FUNCTION_BLOCK FB_Joystick_Input_Scaling
VAR_INPUT
<<<<<<< HEAD
	nRawInput : INT; 
	stJoystickInputScaling : ST_JoystickInputScaling;
	eStatus : E_Status := E_Status.Checking; // bEnable erstatter
=======
	bEnable : BOOL;
	nRawInput : INT; 
	stJoystickInputScaling : ST_JoystickInputScaling;
>>>>>>> 39be3fc96e305d29936f65dffbbc69267e7bf2cf
END_VAR
VAR_OUTPUT
	fNormalizedOutput : LREAL; 
END_VAR
VAR
	fRawInput : LREAL;
	fTempInput : LREAL;
	fTempOutput : LREAL; 
END_VAR

fRawInput := INT_TO_LREAL(nRawInput); // konverterer heltallsverdi fra joystick til flyt-verdi, for beregninger med desimaltall

fTempInput := fRawInput - stJoystickInputScaling.fNeutralInputValue; //Midlertidig variabel før normalisering, midtstilling får en verdi nær 0

IF fTempInput > stJoystickInputScaling.fNeutralDeadband THEN
	fTempOutput := fTempInput/(stJoystickInputScaling.fMaxInputValue - stJoystickInputScaling.fNeutralInputValue);	// Normalisert verdi mellom 0 og 1

ELSIF	fTempInput < -stJoystickInputScaling.fNeutralInputValue THEN 
	fTempOutput := fTempInput/(stJoystickInputScaling.fMaxInputValue - stJoystickInputScaling.fNeutralInputValue); // Normalisert vedi mellom 0 og -1
	
ELSE	
    fTempOutput := 0.0;
END_IF

<<<<<<< HEAD
IF eStatus = E_status.Running AND G_IO.bManualSwitch THEN
=======
IF bEnable THEN
>>>>>>> 39be3fc96e305d29936f65dffbbc69267e7bf2cf
	fNormalizedOutput := LIMIT(stJoystickInputScaling.fMinOutputValue, fTempOutput, stJoystickInputScaling.fMaxOutputValue); //setter på limit for å forsikre verdien havner mellom -1 og 1
	
ELSE 
	fNormalizedOutput := 0.0;
	
END_IF

END_FUNCTION_BLOCK

(* stored: Version 1.1.0.1
   POU FB_Joystick_Input_Scaling: Id {f799c84b-6800-4554-bc05-8e0cc8249bf6}, SpecialFunc None *)
